FUNCTION_BLOCK FB_Drill IMPLEMENTS I_Drill
VAR
	tProductionTime		: TIME := T#1S; 
	tonProductionPulse 	: TON  ; // productie tick
	cProducedProducts :  CTUD := (PV := 100) ; // total units produced
END_VAR

// production tick
tonProductionPulse(pt := tProductionTime , IN := NOT tonProductionPulse.Q);
// produce part
cProducedProducts.RESET := FALSE;
cProducedProducts.CU := tonProductionPulse.Q;

{warning 'Add property implementation'}
PROPERTY ProductsOut : UINT
GET
ProductsOut := cProducedProducts.CV;
cProducedProducts.RESET := TRUE;
END_GET
END_PROPERTY

END_FUNCTION_BLOCK

(* stored: Version 1.1.0.1, ProductVersion 3.1.4024.13
   POU FB_Drill: Id {4a272c19-a7a2-41f9-ab02-d976772d0eef}, SpecialFunc None
   Property ProductsOut: Id {9afa9b60-be3b-430f-bb61-66cafa15a896}
   Get Get: Id {8ddbff59-4e9c-4c09-9e21-4ad225626140} *)
